// TwinCAT 3 PLC project PISTON_TEST
// ProgramVersion: 3.1.4023.0
// libraries:
//   Tc2_Standard, * (Beckhoff Automation GmbH)
//   Tc2_System, * (Beckhoff Automation GmbH)
//   Tc2_Utilities, * (Beckhoff Automation GmbH)
//   Tc3_Module, * (Beckhoff Automation GmbH)
// project tree:
//   DUTs/ ePistonStatus.TcDUT, E_CONVAYOR_STATE.TcDUT, E_MAIN_STATE.TcDUT, E_PISTON_STATE.TcDUT, E_PISTON_TYPE.TcDUT (not stored), E_STATION_STATE.TcDUT, ST_CART.TcDUT, ST_PISTON.TcDUT
//   GVLs/ GVL.TcGVL
//   / PlcTask.TcTTO
//   POUs/ CLEAN.TcPOU, FB_SEPARATE.TcPOU, MAIN_CONVAYOR.TcPOU, FB_CART.TcPOU, FB_NEW_PISTON.TcPOU, MAIN.TcPOU, PISTONS_CYCLE.TcPOU, SUPPLY.TcPOU, SUPPLY_CONVAYOR.TcPOU (not stored), UpdateTimeStamp.TcPOU (not stored)
// real-time tasks:
//   TASK PlcTask: cycle T#10ms, priority 20, ADS port 350
// motion (NC):
//   TASK NC-Task 1 SAF: cycle T#2ms, priority 4, ADS port 501
//   TASK NC-Task 1 SVB: cycle T#10ms, priority 8, ADS port 511
//   AXIS MAIN (id 1)
//     OtherSettings: AllowMotionCmdToSlave=true
//     encoder EncType=19
//       EncPara: MaxCount=#xffffffff
//     drive DrvType=16
//       DrvPara: MaxCount=#xffffffff, DriveControlDWord=#x00000100
//         Analog: TorqueSetpointScale=10, ScaleFactorActTorque=0.1
//         TimeComp: TaskDelayCycles=1
//     controller CtrType=1
//       CtrPara: PriorControlFactor=1
//         Observer: BandWidth=20
//   AXIS SUPPLY (id 2)
//     OtherSettings: AllowMotionCmdToSlave=true
//     encoder EncType=19
//       EncPara: MaxCount=#xffffffff
//     drive DrvType=16
//       DrvPara: MaxCount=#xffffffff, DriveControlDWord=#x00000100
//         Analog: TorqueSetpointScale=10, ScaleFactorActTorque=0.1
//         TimeComp: TaskDelayCycles=1
//     controller CtrType=1
//       CtrPara: PriorControlFactor=1
//         Observer: BandWidth=20
//   AXIS JACK1 (id 3)
//     OtherSettings: AllowMotionCmdToSlave=true
//     encoder EncType=1
//     drive DrvType=5
//       Analog: TorqueSetpointScale=10, ScaleFactorActTorque=0.1
//       TimeComp: TaskDelayCycles=1
//     controller CtrType=1
//       CtrPara: PriorControlFactor=1
//         Observer: BandWidth=20
//   AXIS JACK2 (id 4)
//     OtherSettings: AllowMotionCmdToSlave=true
//     encoder EncType=1
//     drive DrvType=5
//       Analog: TorqueSetpointScale=10, ScaleFactorActTorque=0.1
//     controller CtrType=1
//       CtrPara: PriorControlFactor=1
//         Observer: BandWidth=20
// I/O:
//   DEVICE Device 3 (EtherCAT), AmsNetId 5.109.70.127.4.1
//     Term 1 (EK1100) [EK1100 EtherCAT Coupler (2A E-Bus)]
//       Term 2 (EL1809) [EL1809 16Ch. Dig. Input 24V, 3ms]
//       Term 10 (EL1809) [EL1809 16Ch. Dig. Input 24V, 3ms]
//       Term 11 (EL1809) [EL1809 16Ch. Dig. Input 24V, 3ms]
//       Term 13 (EL1809) [EL1809 16Ch. Dig. Input 24V, 3ms]
//       Term 3 (EL2869) [EL2869 16Ch. Dig Output 24V, 0.5A, Diagnostic]
//       Term 4 (EL6224) [EL6224 (IO Link Master)]
//       Term 15 (EL9011) [EL9011 End Terminal]
//       Term 7 (EL9011) [EL9011 End Terminal]
//     MAIN
//     SUPPLY [CD02 EtherCAT Drive (CoE)]
// variable links:
//   (this object) <-> Device 3 (EtherCAT)/MAIN
//     Drive/Inputs/In/nDataIn1 <-> TxPDO 1/Following Error Actual Value
//     Drive/Inputs/In/nDataIn3[0] <-> TxPDO 4/Torque Actual Value
//     Drive/Inputs/In/nDcOutputTime <-> InfoData/DcOutputShift
//     Drive/Inputs/In/nState1 <-> TxPDO 4/Statusword
//     Drive/Inputs/In/nState2 <-> TxPDO 4/Statusword @bit 8
//     Drive/Inputs/In/nState4 @bit 1 <-> WcState/InputToggle
//     Drive/Inputs/In/nState4 <-> WcState/WcState
//     Drive/Inputs/In/nState5 <-> TxPDO 3/Modes of Operation Display
//     Drive/Outputs/Out/nCtrl1 <-> RxPDO 4/Controlword
//     Drive/Outputs/Out/nCtrl2 <-> RxPDO 4/Controlword @bit 8
//     Drive/Outputs/Out/nCtrl5 <-> RxPDO 4/Modes of Operation
//     Drive/Outputs/Out/nDataOut1 <-> RxPDO 1/Target Position
//     Drive/Outputs/Out/nDataOut2 <-> RxPDO 2/Target Velocity
//     Drive/Outputs/Out/nDataOut3[0] <-> RxPDO 4/Torque Offset
//     Drive/Outputs/Out/nDataOut4[0] <-> RxPDO 3/Target Torque
//     Enc/Inputs/In/nDataIn1 <-> TxPDO 2/Position Actual Value
//     Enc/Inputs/In/nDcInputTime <-> InfoData/DcInputShift
//     Enc/Inputs/In/nState4 @bit 1 <-> WcState/InputToggle
//     Enc/Inputs/In/nState4 <-> WcState/WcState
//   (this object) <-> Device 3 (EtherCAT)/SUPPLY
//     Drive/Inputs/In/nDataIn1 <-> TxPDO 1/Following Error Actual Value
//     Drive/Inputs/In/nDataIn3[0] <-> TxPDO 4/Torque Actual Value
//     Drive/Inputs/In/nDcOutputTime <-> InfoData/DcOutputShift
//     Drive/Inputs/In/nState1 <-> TxPDO 4/Statusword
//     Drive/Inputs/In/nState2 <-> TxPDO 4/Statusword @bit 8
//     Drive/Inputs/In/nState4 @bit 1 <-> WcState/InputToggle
//     Drive/Inputs/In/nState4 <-> WcState/WcState
//     Drive/Inputs/In/nState5 <-> TxPDO 3/Modes of Operation Display
//     Drive/Outputs/Out/nCtrl1 <-> RxPDO 4/Controlword
//     Drive/Outputs/Out/nCtrl2 <-> RxPDO 4/Controlword @bit 8
//     Drive/Outputs/Out/nCtrl5 <-> RxPDO 4/Modes of Operation
//     Drive/Outputs/Out/nDataOut1 <-> RxPDO 1/Target Position
//     Drive/Outputs/Out/nDataOut2 <-> RxPDO 2/Target Velocity
//     Drive/Outputs/Out/nDataOut3[0] <-> RxPDO 4/Torque Offset
//     Drive/Outputs/Out/nDataOut4[0] <-> RxPDO 3/Target Torque
//     Enc/Inputs/In/nDataIn1 <-> TxPDO 2/Position Actual Value
//     Enc/Inputs/In/nDcInputTime <-> InfoData/DcInputShift
//     Enc/Inputs/In/nState4 @bit 1 <-> WcState/InputToggle
//     Enc/Inputs/In/nState4 <-> WcState/WcState
//   TAMAR_22mm Instance <-> Device 3 (EtherCAT)/Term 1 (EK1100)/Term 2 (EL1809)
//     PlcTask Inputs/GVL_IO.inputs[1]/ch{1..16} <-> Channel {1..16}/ch{1..16}  (16 links)
//   TAMAR_22mm Instance <-> Device 3 (EtherCAT)/Term 1 (EK1100)/Term 3 (EL2869)
//     PlcTask Outputs/GVL_IO.outputs[1]/ch{1..16} <-> DOS Outputs Channel {1..16}/Output  (16 links)
//   TAMAR_22mm Instance <-> Device 3 (EtherCAT)/Term 1 (EK1100)/Term 4 (EL6224)
//     PlcTask Outputs/GVL_IO.uIOLINK1 <-> IO-Link Port1_out/GVL_IO.uIOLINK1
//     PlcTask Outputs/GVL_IO.uIOLINK2 <-> IO-Link Port2_out/GVL_IO.uIOLINK2
//   TAMAR_22mm Instance <-> NC-Task 1 SAF/Axes/JACK1
//     PlcTask Inputs/GVL.Axis_JACK1.Axis.NcToPlc <-> Outputs/ToPlc
//     PlcTask Outputs/GVL.Axis_JACK1.Axis.PlcToNc <-> Inputs/FromPlc
//   TAMAR_22mm Instance <-> NC-Task 1 SAF/Axes/JACK2
//     PlcTask Inputs/GVL.Axis_JACK2.Axis.NcToPlc <-> Outputs/ToPlc
//     PlcTask Outputs/GVL.Axis_JACK2.Axis.PlcToNc <-> Inputs/FromPlc
//   TAMAR_22mm Instance <-> NC-Task 1 SAF/Axes/MAIN
//     PlcTask Inputs/GVL.Axis_MAIN.Axis.NcToPlc <-> Outputs/ToPlc
//     PlcTask Outputs/GVL.Axis_MAIN.Axis.PlcToNc <-> Inputs/FromPlc
//   TAMAR_22mm Instance <-> NC-Task 1 SAF/Axes/SUPPLY
//     PlcTask Inputs/GVL.Axis_SUPPLY.Axis.NcToPlc <-> Outputs/ToPlc
//     PlcTask Outputs/GVL.Axis_SUPPLY.Axis.PlcToNc <-> Inputs/FromPlc

CONFIGURATION PISTON_TEST
    RESOURCE PLC ON TwinCAT3
        TASK PlcTask(INTERVAL := T#10ms, PRIORITY := 20);
        PROGRAM MAIN WITH PlcTask : MAIN;
    END_RESOURCE
END_CONFIGURATION

// ---- DUTs/ePistonStatus.TcDUT
{attribute 'qualified_only'}
{attribute 'strict'}
TYPE ePistonStatus :
(
	OPENED:=0,CLOSED,OPENING,CLOSING,ERROR
);
END_TYPE

// ---- DUTs/E_CONVAYOR_STATE.TcDUT
{attribute 'qualified_only'}
{attribute 'strict'}
TYPE E_CONVAYOR_STATE :
(
	uninit,
	idle,
	do_move,
	done,
	pause,
	error
);
END_TYPE

// ---- DUTs/E_MAIN_STATE.TcDUT
{attribute 'qualified_only'}
{attribute 'strict'}
TYPE E_MAIN_STATE :
(
	uninit,
	idle,
	do_actions,
	move_next,
	done,
	pause,
	error
);
END_TYPE

// ---- DUTs/E_PISTON_STATE.TcDUT
{attribute 'qualified_only'}
{attribute 'strict'}
TYPE E_PISTON_STATE :
(
	init,
	ready,
	busy,
	done,
	error
);
END_TYPE

// ---- DUTs/E_STATION_STATE.TcDUT
{attribute 'qualified_only'}
{attribute 'strict'}
TYPE E_STATION_STATE :
(
	uninit,
	idle,
	do_action1,
	do_action2,
	do_action3,
	do_action4,
	do_action5,
	done,
	pause,
	error
);
END_TYPE

// ---- DUTs/ST_CART.TcDUT
TYPE ST_CART :
STRUCT
	nNAME: STRING;
	posX:INT;
	posY:INT;
	color:INT;
	position: INT;
END_STRUCT
END_TYPE

// ---- DUTs/ST_PISTON.TcDUT
TYPE ST_PISTON :
STRUCT
	ePISTON_TYPE: E_PISTON_TYPE;
	
	nNAME: STRING;
	openTime: REAL:=5;
	closeTime: REAL:=5;
	timeoutOpen:  TIME:=T#5S;
	timeoutClose: TIME:=T#5S;
	bOPEN_BY_DEFAULT: BOOL:= FALSE;
END_STRUCT
	
END_TYPE

// ---- GVLs/GVL.TcGVL
 //{attribute 'qualified_only'}
VAR_GLOBAL
	
	supply_station_num: INT:=1;
	separate1_station_num: INT:=5;
	separate2_station_num: INT:=9;
	clean_station_num: INT:=24;
	total_ready:INT:=0;
	iNUMBER_OF_PISTONS: INT:=15;
	conv_length: INT:=1150;
	conv_height: INT:=290;
	num_of_carts:INT:=18;
	X_OFFSET: INT:=380;
	Y_OFFSET: INT:=352;
	stPISTON_PARAM: ARRAY[1..15] OF  ST_PISTON;
	fbPiston: ARRAY[1..15] OF FB_NEW_PISTON;
	fbCART: ARRAY[1..18] OF FB_CART;
	posArrX:ARRAY[1..36] OF INT;
	posArrY:ARRAY[1..36] OF INT;
	
	eMAIN_STATE: E_MAIN_STATE:= E_MAIN_STATE.uninit;
	eSUPPLY: E_STATION_STATE:=E_STATION_STATE.uninit;
	eSEPARATE1: E_STATION_STATE:=E_STATION_STATE.uninit;
	eSEPARATE2: E_STATION_STATE:=E_STATION_STATE.uninit;
	eCLEAN: E_STATION_STATE:=E_STATION_STATE.uninit;
	eMAIN_CONVAYOR_STATE: E_CONVAYOR_STATE:=E_CONVAYOR_STATE.uninit;
	eSUPPLY_CONVAYOR_STATE: E_CONVAYOR_STATE:=E_CONVAYOR_STATE.uninit;
	
	bSTART: BOOL:=FALSE;// start main state machine
	sup_RUNNING: BOOL:=FALSE;// supply id runing
	clean_RUNNING: BOOL:=FALSE;// cleaning runing
	bS1_RUNNING: BOOL:=FALSE; // station 1 is running
	bS2_RUNNING: BOOL:=FALSE; // station 2 is running
	bCONV_MAIN_INPOS: BOOL:=FALSE; // convayor in position
	bCONV_SUPPLY_INPOS: BOOL:=FALSE; // convayor in position
	bPAUSE_MAIN: BOOL:=FALSE;
	
	
END_VAR

// ---- POUs/MAIN.TcPOU
PROGRAM MAIN
VAR
	counter:INT:=0;
	iNUMBER1 : INT:=2;
	sNAME1 : STRING(255):='24_5A';
	Trigger : BOOL;
	rtrigSTART: R_TRIG;
	rtrigPAUSE: R_TRIG;
	ftrigRERUN: F_TRIG;
	temp_state:E_MAIN_STATE;
	temp_supply_state:E_STATION_STATE;
	temp_sep1_state:E_STATION_STATE;
	temp_sep2_state:E_STATION_STATE;
	temp_clean_state:E_STATION_STATE;
	temp_conv_state:E_CONVAYOR_STATE;
	temp_supconv_state:E_CONVAYOR_STATE;
	
	fbSEPARATION1: FB_SEPARATE;		
	fbSEPARATION2: FB_SEPARATE;	
	
	action_timeout: TON:=(PT:=T#20s);
	move_timeout: TON;
	bTIMEOUT:BOOL:=FALSE;
END_VAR

A_ERROR_CHECK();
PISTONS_CYCLE();
MAIN_CONVAYOR();
SUPPLY_CONVAYOR();
SUPPLY();
fbSEPARATION1(piston_updown:=  fbPiston[3],
			  piston_colet:=  fbPiston[4],
			  piston_puller:=  fbPiston[5],
			  piston_tray:=  fbPiston[6],
			  piston_pins:=  fbPiston[7],
			  eState:= eSEPARATE1 );
		
fbSEPARATION2(piston_updown:=  fbPiston[8],
			  piston_colet:=  fbPiston[9],
			  piston_puller:=  fbPiston[10],
			  piston_tray:=  fbPiston[11],
			  piston_pins:=  fbPiston[12],
			  eState:= eSEPARATE2 );	
	
CLEAN();

rtrigSTART(CLK:= bSTART, Q=> );
rtrigPAUSE(CLK:= bPAUSE_MAIN, Q=> );
ftrigRERUN(CLK:= bPAUSE_MAIN, Q=> );
action_timeout(IN:=bTIMEOUT);

//MAIN_STATE_MACHINE:
CASE eMAIN_STATE OF
	E_MAIN_STATE.uninit:
		bTIMEOUT:=FALSE;
		IF rtrigSTART.Q THEN
			eMAIN_STATE:=E_MAIN_STATE.do_actions;
		END_IF
	
	E_MAIN_STATE.do_actions:
		bTIMEOUT:=TRUE;
		IF eSUPPLY = E_STATION_STATE.idle THEN     
			eSUPPLY := E_STATION_STATE.do_action1;
		END_IF
		IF eSEPARATE1 = E_STATION_STATE.idle THEN
			eSEPARATE1 := E_STATION_STATE.do_action1;
		END_IF
		IF eSEPARATE2 = E_STATION_STATE.idle THEN
			eSEPARATE2 := E_STATION_STATE.do_action1;
		END_IF
		IF eCLEAN = E_STATION_STATE.idle THEN
			eCLEAN := E_STATION_STATE.do_action1;
		END_IF
		
		IF (eSEPARATE1 = E_STATION_STATE.done AND eSEPARATE2 = E_STATION_STATE.done AND eSUPPLY = E_STATION_STATE.done  AND eCLEAN = E_STATION_STATE.done) THEN
			eSUPPLY := E_STATION_STATE.idle;
			eSEPARATE1 := E_STATION_STATE.idle;
			eSEPARATE2 := E_STATION_STATE.idle;
			eCLEAN := E_STATION_STATE.idle;
			eMAIN_STATE:=E_MAIN_STATE.move_next;
			bTIMEOUT:=FALSE;
		END_IF
		
		IF action_timeout.Q THEN
			eMAIN_STATE:=E_MAIN_STATE.error;
		END_IF
		
	E_MAIN_STATE.move_next: 
		IF eMAIN_CONVAYOR_STATE = E_CONVAYOR_STATE.idle THEN
			eMAIN_CONVAYOR_STATE := E_CONVAYOR_STATE.do_move;
		END_IF
		IF eSUPPLY_CONVAYOR_STATE = E_CONVAYOR_STATE.idle THEN
			eSUPPLY_CONVAYOR_STATE := E_CONVAYOR_STATE.do_move;
		END_IF
		IF eMAIN_CONVAYOR_STATE = E_CONVAYOR_STATE.done AND eSUPPLY_CONVAYOR_STATE = E_CONVAYOR_STATE.done THEN
			eMAIN_CONVAYOR_STATE := E_CONVAYOR_STATE.idle;
			eSUPPLY_CONVAYOR_STATE := E_CONVAYOR_STATE.idle;
			eMAIN_STATE:=E_MAIN_STATE.do_actions;
		END_IF
		
	E_MAIN_STATE.pause: 
		bTIMEOUT:=FALSE;
		//paused
		
	E_MAIN_STATE.error: 
		//error mode

END_CASE

IF rtrigPAUSE.Q THEN
	temp_state:=eMAIN_STATE;
	temp_supply_state:=eSUPPLY;
	temp_sep1_state:=eSEPARATE1;
	temp_sep2_state:=eSEPARATE2;
	temp_clean_state:=eCLEAN;
	temp_conv_state:=eMAIN_CONVAYOR_STATE;
	temp_supconv_state:=eMAIN_CONVAYOR_STATE;
	eMAIN_STATE:=E_MAIN_STATE.pause;
	eSUPPLY:=E_STATION_STATE.pause;
	eSEPARATE1:=E_STATION_STATE.pause;
	eSEPARATE2:=E_STATION_STATE.pause;
	eMAIN_CONVAYOR_STATE:=E_CONVAYOR_STATE.pause;
	eSUPPLY_CONVAYOR_STATE:=E_CONVAYOR_STATE.pause;
	
END_IF

IF ftrigRERUN.Q THEN
	eMAIN_STATE:=temp_state;
	eSUPPLY:=temp_supply_state;
	eSEPARATE1:=temp_sep1_state;
	eSEPARATE2:=temp_sep2_state;
	eCLEAN:=temp_clean_state;
	eMAIN_CONVAYOR_STATE:=temp_conv_state;
	eSUPPLY_CONVAYOR_STATE:=temp_conv_state;
END_IF

ACTION A_ERROR_CHECK:
FOR counter:=1 TO iNUMBER_OF_PISTONS BY 1 DO
	IF fbPiston[counter].PistonStatus = ePistonStatus.ERROR THEN
		eMAIN_STATE:=E_MAIN_STATE.error;
		
	END_IF
	
END_FOR;
END_ACTION

END_PROGRAM

// ---- POUs/FB_SEPARATE.TcPOU
FUNCTION_BLOCK FB_SEPARATE
VAR_INPUT
	piston_updown: REFERENCE TO FB_NEW_PISTON;
	piston_colet: REFERENCE TO FB_NEW_PISTON;
	piston_puller: REFERENCE TO FB_NEW_PISTON;
	piston_tray: REFERENCE TO FB_NEW_PISTON;
	piston_pins: REFERENCE TO FB_NEW_PISTON;
	eState: REFERENCE TO  E_STATION_STATE;
END_VAR
VAR_OUTPUT
	bRUNNING:BOOL :=FALSE;
END_VAR
VAR
	tDelay: TON;
	bDELAY: BOOL:=FALSE;
	E: INT;
END_VAR

tDelay(IN:=bDELAY);

CASE eState OF
	E_STATION_STATE.uninit:
		eState:= E_STATION_STATE.idle;

	E_STATION_STATE.idle:
		bRUNNING:=FALSE;
			

	E_STATION_STATE.do_action1://delay and lower device
		bRUNNING:=TRUE;
		tDELAY.PT:=T#0.1S;
		bDELAY:=TRUE;
		IF tDELAY.Q THEN
			bDELAY:=FALSE;
			piston_updown.A_OPEN();
		END_IF
		
		IF piston_updown.PistonStatus= ePistonStatus.OPENED THEN
			eState:=E_STATION_STATE.do_action2;
		END_IF
		
	E_STATION_STATE.do_action2://delay and close colet
		tDELAY.PT:=T#0.1S;
		bDELAY:=TRUE;
		IF tDELAY.Q THEN
			bDELAY:=FALSE;
			piston_colet.A_OPEN();
		END_IF
		
		IF piston_colet.PistonStatus= ePistonStatus.OPENED THEN
			eState:=E_STATION_STATE.do_action3;
		END_IF
	
	E_STATION_STATE.do_action3://delay and pull while raising
		tDELAY.PT:=T#0.2S;		
		bDELAY:=TRUE;
		IF tDELAY.Q THEN
			bDELAY:=FALSE;
			piston_updown.A_CLOSE();
			piston_puller.A_OPEN();
		END_IF
		IF piston_updown.PistonStatus= ePistonStatus.CLOSED AND piston_puller.PistonStatus= ePistonStatus.OPENED THEN
			eState:=E_STATION_STATE.do_action4;
		END_IF
	
	E_STATION_STATE.do_action4://delay close puller and enter tray
		tDELAY.PT:=T#0.2S;		
		bDELAY:=TRUE;
		IF tDELAY.Q THEN
			bDELAY:=FALSE;
			piston_puller.A_CLOSE();
			piston_tray.A_OPEN();
		END_IF
		IF piston_puller.PistonStatus= ePistonStatus.CLOSED AND piston_tray.PistonStatus= ePistonStatus.OPENED THEN
			eState:=E_STATION_STATE.do_action5;
		END_IF

	E_STATION_STATE.do_action5://release colet and push pins
		tDELAY.PT:=T#0.2S;		
		bDELAY:=TRUE;
		IF tDELAY.Q THEN
			bDELAY:=FALSE;
			piston_colet.A_CLOSE();
			piston_pins.A_OPEN();
		END_IF
		IF piston_colet.PistonStatus= ePistonStatus.CLOSED AND piston_pins.PistonStatus= ePistonStatus.OPENED THEN
			eState:=E_STATION_STATE.do_action6;
		END_IF
		
	E_STATION_STATE.do_action6://raise pins and close tray
		tDELAY.PT:=T#0.2S;		
		bDELAY:=TRUE;
		IF tDELAY.Q THEN
			bDELAY:=FALSE;
			piston_pins.A_CLOSE();
			piston_tray.A_CLOSE();
		END_IF
		IF piston_colet.PistonStatus= ePistonStatus.CLOSED AND piston_pins.PistonStatus= ePistonStatus.CLOSED THEN
			eState:=E_STATION_STATE.do_action7;
		END_IF	
		
	E_STATION_STATE.do_action7://delay
		tDELAY.PT:=T#0.1S;
		bDELAY:=TRUE;
		IF tDELAY.Q THEN
			bDELAY:=FALSE;
			eState:=E_STATION_STATE.done;
		END_IF
		
	
	E_STATION_STATE.done:
		bRUNNING:=FALSE;
		
	E_STATION_STATE.pause:
		//paused

END_CASE

END_FUNCTION_BLOCK

// ---- POUs/FB_NEW_PISTON.TcPOU
FUNCTION_BLOCK FB_NEW_PISTON
VAR_INPUT
	
	bMANUAL:BOOL:=FALSE;
	stPISTON:   ST_PISTON;
	bCMD_OPEN_SWR: BOOL;
	bCMD_CLOSE_SWR: BOOL;
	bCMD_OPEN: BOOL;
	bSEN_OPEN: BOOL;
	bSEN_CLOSE: BOOL;
END_VAR
VAR_OUTPUT
	PistonStatus:ePistonStatus;
	bVALVE_OPEN: BOOL;
	bVALVE_CLOSE: BOOL;
	
	
END_VAR
VAR
	timerOpening:ton;
	timerClosing:ton;
	timeoutOpening:ton;
	timeoutClosing:ton;
	bSTARTUP: BOOL:=FALSE;
	
	
END_VAR

   IF NOT bSTARTUP THEN
	bCMD_OPEN:=stPISTON.bOPEN_BY_DEFAULT;
	bSTARTUP:=TRUE;
END_IF

timerOpening(IN:= bVALVE_OPEN, PT:=REAL_TO_TIME(stPISTON.openTime)*1000 , Q=> , ET=> );
timerClosing(IN:= NOT bVALVE_OPEN, PT:=REAL_TO_TIME(stPISTON.closeTime)*1000 , Q=> , ET=> );
timeoutOpening(IN:= bVALVE_OPEN AND NOT bSEN_OPEN, PT:= stPISTON.timeoutOpen, Q=> , ET=> );
timeoutClosing(IN:= NOT bVALVE_OPEN AND NOT bSEN_CLOSE, PT:= stPISTON.timeoutClose, Q=> , ET=> );
IF bMANUAL THEN
	bVALVE_OPEN:= bCMD_OPEN;
	bVALVE_CLOSE:= NOT bCMD_OPEN;
ELSE
	bVALVE_OPEN:= bCMD_OPEN_SWR;
	bVALVE_CLOSE:= NOT bCMD_OPEN_SWR;
END_IF



CASE stPISTON.ePISTON_TYPE OF
	0://NO_SENSORS
		IF bVALVE_OPEN AND NOT timerOpening.Q THEN
			PistonStatus:=ePistonStatus.OPENING;
		ELSIF bVALVE_OPEN AND timerOpening.Q THEN
			PistonStatus:=ePistonStatus.OPENED;
		ELSIF bVALVE_CLOSE AND NOT timerClosing.Q THEN
			PistonStatus:=ePistonStatus.CLOSING;
		ELSIF bVALVE_CLOSE AND timerClosing.Q THEN
			PistonStatus:=ePistonStatus.CLOSED;
		END_IF
		
 
	
	1://only open sensor
	
		IF bVALVE_OPEN AND NOT bSEN_OPEN THEN
			PistonStatus:=ePistonStatus.OPENING;
		ELSIF bVALVE_OPEN AND bSEN_OPEN THEN
			PistonStatus:=ePistonStatus.OPENED;
		ELSIF bVALVE_CLOSE AND NOT timerClosing.Q THEN
			PistonStatus:=ePistonStatus.CLOSING;
		ELSIF bVALVE_CLOSE AND timerClosing.Q THEN
			PistonStatus:=ePistonStatus.CLOSED;
		END_IF
	
	2:// only close sensor
		IF bVALVE_OPEN AND NOT timerOpening.Q THEN
			PistonStatus:=ePistonStatus.OPENING;
		ELSIF bVALVE_OPEN AND timerOpening.Q THEN
			PistonStatus:=ePistonStatus.OPENED;
		ELSIF bVALVE_CLOSE AND NOT bSEN_CLOSE THEN
			PistonStatus:=ePistonStatus.CLOSING;
		ELSIF bVALVE_CLOSE AND bSEN_CLOSE THEN
			PistonStatus:=ePistonStatus.CLOSED;
		END_IF
	
	
	3://both sensors
		IF bVALVE_OPEN AND NOT bSEN_OPEN THEN
			PistonStatus:=ePistonStatus.OPENING;
		ELSIF bVALVE_OPEN AND bSEN_OPEN THEN
			PistonStatus:=ePistonStatus.OPENED;
		ELSIF bVALVE_CLOSE AND NOT bSEN_CLOSE THEN
			PistonStatus:=ePistonStatus.CLOSING;
		ELSIF bVALVE_CLOSE AND bSEN_CLOSE THEN
			PistonStatus:=ePistonStatus.CLOSED;
		END_IF
	
END_CASE

IF timeoutOpening.Q AND (stPISTON.ePISTON_TYPE = E_PISTON_TYPE.ONLY_OPEN OR stPISTON.ePISTON_TYPE = E_PISTON_TYPE.BOTH)  THEN
	PistonStatus:=ePistonStatus.ERROR;
END_IF
IF timeoutClosing.Q  AND (stPISTON.ePISTON_TYPE = E_PISTON_TYPE.ONLY_CLOSE OR stPISTON.ePISTON_TYPE = E_PISTON_TYPE.BOTH)  THEN
	PistonStatus:=ePistonStatus.ERROR;
END_IF

ACTION A_CLOSE:
bCMD_OPEN_SWR:=FALSE;
END_ACTION

ACTION A_OPEN:
bCMD_OPEN_SWR:=TRUE;
END_ACTION

END_FUNCTION_BLOCK

// ---- POUs/PISTONS_CYCLE.TcPOU
PROGRAM PISTONS_CYCLE
VAR
	
	bSTARTUP: BOOL:=FALSE;
	counter: INT;
	
END_VAR

IF NOT bSTARTUP THEN
	
	stPISTON_PARAM[1].nNAME:='SUPPLY 1';
	stPISTON_PARAM[1].bOPEN_BY_DEFAULT:=FALSE;
	stPISTON_PARAM[1].openTime:=0.2;
	stPISTON_PARAM[1].closeTime:=0.2;
	stPISTON_PARAM[1].timeoutOpen:=T#3S;
	stPISTON_PARAM[1].timeoutClose:=T#3S;
	stPISTON_PARAM[1].ePISTON_TYPE:= 0;

	stPISTON_PARAM[2].nNAME:='SUPPLY2';
	stPISTON_PARAM[2].bOPEN_BY_DEFAULT:=FALSE;
	stPISTON_PARAM[2].openTime:=0.2;
	stPISTON_PARAM[2].closeTime:=0.2;
	stPISTON_PARAM[2].timeoutOpen:=T#2S;
	stPISTON_PARAM[2].timeoutClose:=T#2S;
	stPISTON_PARAM[2].ePISTON_TYPE:= 0;

	stPISTON_PARAM[3].nNAME:='SEPARATE1 UP_DOWN';
	stPISTON_PARAM[3].bOPEN_BY_DEFAULT:=FALSE;
	stPISTON_PARAM[3].openTime:=0.2;
	stPISTON_PARAM[3].closeTime:=0.2;
	stPISTON_PARAM[3].timeoutOpen:=T#3S;
	stPISTON_PARAM[3].timeoutClose:=T#3S;
	stPISTON_PARAM[3].ePISTON_TYPE:= 0;
	
	stPISTON_PARAM[4].nNAME:='SEPARATE1 COLET';
	stPISTON_PARAM[4].bOPEN_BY_DEFAULT:=FALSE;
	stPISTON_PARAM[4].openTime:=0.2;
	stPISTON_PARAM[4].closeTime:=0.2;
	stPISTON_PARAM[4].timeoutOpen:=T#3S;
	stPISTON_PARAM[4].timeoutClose:=T#3S;
	stPISTON_PARAM[4].ePISTON_TYPE:= 0;
	
	stPISTON_PARAM[5].nNAME:='SEPARATE1 PULL';
	stPISTON_PARAM[5].bOPEN_BY_DEFAULT:=FALSE;
	stPISTON_PARAM[5].openTime:=0.2;
	stPISTON_PARAM[5].closeTime:=0.2;
	stPISTON_PARAM[5].timeoutOpen:=T#3S;
	stPISTON_PARAM[5].timeoutClose:=T#3S;
	stPISTON_PARAM[5].ePISTON_TYPE:= 0;
	
	stPISTON_PARAM[6].nNAME:='SEPARATE1 TRAY';
	stPISTON_PARAM[6].bOPEN_BY_DEFAULT:=FALSE;
	stPISTON_PARAM[6].openTime:=0.2;
	stPISTON_PARAM[6].closeTime:=0.2;
	stPISTON_PARAM[6].timeoutOpen:=T#3S;
	stPISTON_PARAM[6].timeoutClose:=T#3S;
	stPISTON_PARAM[6].ePISTON_TYPE:= 0;
	
	stPISTON_PARAM[7].nNAME:='SEPARATE1 PINS';
	stPISTON_PARAM[7].bOPEN_BY_DEFAULT:=FALSE;
	stPISTON_PARAM[7].openTime:=0.2;
	stPISTON_PARAM[7].closeTime:=0.2;
	stPISTON_PARAM[7].timeoutOpen:=T#3S;
	stPISTON_PARAM[7].timeoutClose:=T#3S;
	stPISTON_PARAM[7].ePISTON_TYPE:= 0;
	
	stPISTON_PARAM[8].nNAME:='SEPARATE2 UP_DOWN';
	stPISTON_PARAM[8].bOPEN_BY_DEFAULT:=FALSE;
	stPISTON_PARAM[8].openTime:=0.2;
	stPISTON_PARAM[8].closeTime:=0.2;
	stPISTON_PARAM[8].timeoutOpen:=T#3S;
	stPISTON_PARAM[8].timeoutClose:=T#3S;
	stPISTON_PARAM[8].ePISTON_TYPE:= 0;
	
	stPISTON_PARAM[9].nNAME:='SEPARATE2 GRIP';
	stPISTON_PARAM[9].bOPEN_BY_DEFAULT:=FALSE;
	stPISTON_PARAM[9].openTime:=0.2;
	stPISTON_PARAM[9].closeTime:=0.2;
	stPISTON_PARAM[9].timeoutOpen:=T#3S;
	stPISTON_PARAM[9].timeoutClose:=T#3S;
	stPISTON_PARAM[9].ePISTON_TYPE:= 0;
	
	stPISTON_PARAM[10].nNAME:='SEPARATE2 PULL';
	stPISTON_PARAM[10].bOPEN_BY_DEFAULT:=FALSE;
	stPISTON_PARAM[10].openTime:=0.2;
	stPISTON_PARAM[10].closeTime:=0.2;
	stPISTON_PARAM[10].timeoutOpen:=T#3S;
	stPISTON_PARAM[10].timeoutClose:=T#3S;
	stPISTON_PARAM[10].ePISTON_TYPE:= 0;
	
	stPISTON_PARAM[11].nNAME:='SEPARATE2 TRAY';
	stPISTON_PARAM[11].bOPEN_BY_DEFAULT:=FALSE;
	stPISTON_PARAM[11].openTime:=0.2;
	stPISTON_PARAM[11].closeTime:=0.2;
	stPISTON_PARAM[11].timeoutOpen:=T#3S;
	stPISTON_PARAM[11].timeoutClose:=T#3S;
	stPISTON_PARAM[11].ePISTON_TYPE:= 0;
	
	stPISTON_PARAM[12].nNAME:='SEPARATE2 PINS';
	stPISTON_PARAM[12].bOPEN_BY_DEFAULT:=FALSE;
	stPISTON_PARAM[12].openTime:=0.2;
	stPISTON_PARAM[12].closeTime:=0.2;
	stPISTON_PARAM[12].timeoutOpen:=T#3S;
	stPISTON_PARAM[12].timeoutClose:=T#3S;
	stPISTON_PARAM[12].ePISTON_TYPE:= 0;
	
	stPISTON_PARAM[13].nNAME:='ADVANCE';
	stPISTON_PARAM[13].bOPEN_BY_DEFAULT:=FALSE;
	stPISTON_PARAM[13].openTime:=0.5;
	stPISTON_PARAM[13].closeTime:=0.5;
	stPISTON_PARAM[13].timeoutOpen:=T#3S;
	stPISTON_PARAM[13].timeoutClose:=T#3S;
	stPISTON_PARAM[13].ePISTON_TYPE:= 0;
	
	stPISTON_PARAM[14].nNAME:='CLEAN';
	stPISTON_PARAM[14].bOPEN_BY_DEFAULT:=FALSE;
	stPISTON_PARAM[14].openTime:=0.2;
	stPISTON_PARAM[14].closeTime:=0.2;
	stPISTON_PARAM[14].timeoutOpen:=T#3S;
	stPISTON_PARAM[14].timeoutClose:=T#3S;
	stPISTON_PARAM[14].ePISTON_TYPE:= 0;
	
	FOR counter:=1 TO iNUMBER_OF_PISTONS BY 1 DO
		fbPiston[counter](stPISTON:=stPISTON_PARAM[counter]);
	END_FOR;
	
	bSTARTUP:=TRUE;
END_IF
FOR counter:=1 TO iNUMBER_OF_PISTONS BY 1 DO
	fbPiston[counter]();
END_FOR;

END_PROGRAM

// ---- POUs/SUPPLY.TcPOU
PROGRAM SUPPLY
VAR

	tDelay: TON;
	bDELAY: BOOL:=FALSE;
END_VAR

tDelay(IN:=bDELAY);
CASE eSUPPLY OF
	E_STATION_STATE.uninit:
		eSUPPLY:= E_STATION_STATE.idle;

	E_STATION_STATE.idle:
		bS1_RUNNING:=FALSE;
			

	E_STATION_STATE.do_action1://delay and open piston1,2
		tDELAY.PT:=T#1S;
		bDELAY:=TRUE;
		IF tDELAY.Q THEN
			bDELAY:=FALSE;
			fbPISTON[1].A_OPEN();
			fbPISTON[2].A_OPEN();
		END_IF
		
		IF fbPISTON[1].PistonStatus= ePistonStatus.OPENED  AND fbPISTON[2].PistonStatus= ePistonStatus.OPENED THEN
			eSUPPLY:=E_STATION_STATE.do_action2;
		END_IF
		
	E_STATION_STATE.do_action2://delay and close pistons 1,2
		tDELAY.PT:=T#2S;		
		bDELAY:=TRUE;
		IF tDELAY.Q THEN
			bDELAY:=FALSE;
			fbPISTON[1].A_CLOSE();
			fbPISTON[2].A_CLOSE();
		END_IF
		IF fbPISTON[1].PistonStatus= ePistonStatus.CLOSED  AND fbPISTON[2].PistonStatus= ePistonStatus.CLOSED THEN
			eSUPPLY:=E_STATION_STATE.do_action5;
		END_IF
	
	E_STATION_STATE.do_action3://delay and open piston 3
		//...
	
	E_STATION_STATE.do_action4://delay and close pistons 1,2
		//...
		
	E_STATION_STATE.do_action5://delay 
		tDELAY.PT:=T#2S;
		bDELAY:=TRUE;
		IF tDELAY.Q THEN
			bDELAY:=FALSE;
			eSUPPLY:=E_STATION_STATE.done;
		END_IF
	
	E_STATION_STATE.done:
		bS1_RUNNING:=FALSE;
		
	E_STATION_STATE.pause:
		//paused

END_CASE

END_PROGRAM

// ---- POUs/CLEAN.TcPOU
PROGRAM CLEAN
VAR
	tDelay: TON;
	bDELAY: BOOL:=FALSE;
END_VAR

tDelay(IN:=bDELAY);
CASE eCLEAN OF
	E_STATION_STATE.uninit:
		eCLEAN:= E_STATION_STATE.idle;

	E_STATION_STATE.idle:
		clean_RUNNING:=FALSE;
			

	E_STATION_STATE.do_action1://delay and open piston8
		clean_RUNNING:=TRUE;
		tDELAY.PT:=T#0.3S;
		bDELAY:=TRUE;
		IF tDELAY.Q THEN
			bDELAY:=FALSE;
			fbPISTON[14].A_OPEN();
		END_IF
		
		IF fbPISTON[14].PistonStatus= ePistonStatus.OPENED THEN
			eCLEAN:=E_STATION_STATE.do_action2;
		END_IF
		
	
	
	E_STATION_STATE.do_action2://delay and close pistons 8
		tDELAY.PT:=T#1S;		
		bDELAY:=TRUE;
		IF tDELAY.Q THEN
			bDELAY:=FALSE;
			fbPISTON[14].A_CLOSE();
		END_IF
		IF fbPISTON[14].PistonStatus= ePistonStatus.CLOSED  THEN
			eCLEAN:=E_STATION_STATE.do_action3;
		END_IF
	
	E_STATION_STATE.do_action3://delay
		tDELAY.PT:=T#1S;
		bDELAY:=TRUE;
		IF tDELAY.Q THEN
			bDELAY:=FALSE;
			eCLEAN:=E_STATION_STATE.done;
		END_IF
		
	
	E_STATION_STATE.done:
		clean_RUNNING:=FALSE;
		
	E_STATION_STATE.pause:
		//paused

END_CASE

END_PROGRAM

// ---- POUs/MAIN_CONVAYOR.TcPOU
PROGRAM MAIN_CONVAYOR
VAR
	inc: INT:=1;
	temp: INT;
	state: INT:=0;
	total_length: INT;
	cart_space: INT;
	cornerX: INT;
	cornerY: INT;
	bMOVE:BOOL :=FALSE;
	bSTARTUP: BOOL:=FALSE;
	rtrigNext: R_TRIG;
	counter: INT;
	tNext: TON;
	tDelay: TON;
	bDELAY: BOOL:=FALSE;
	first_run: BOOL:=FALSE;
END_VAR

FOR counter:=1 TO num_of_carts BY 1 DO
	fbCART[counter]();
END_FOR;

IF NOT first_run THEN
	A_set_cart_spaces();
	A_SETUP();
	first_run:=TRUE;
END_IF



tDelay(IN:=bDELAY);
tNext(IN:=bMOVE , PT:=T#1S , Q=> , ET=> );

CASE eMAIN_CONVAYOR_STATE OF
	E_CONVAYOR_STATE.uninit:
		A_SETUP();
		eMAIN_CONVAYOR_STATE:=E_CONVAYOR_STATE.idle;
	
	E_CONVAYOR_STATE.idle:
		bDELAY:=FALSE;
		bMOVE:=FALSE;
		bCONV_MAIN_INPOS:=TRUE;
	
	E_CONVAYOR_STATE.do_move: // open advance piston and update carts
		IF bCONV_MAIN_INPOS THEN		 
			A_CARTS_STEP();
			fbPISTON[11].A_OPEN();
			bCONV_MAIN_INPOS:=FALSE;
		END_IF
		bMOVE:=TRUE;
		bCONV_MAIN_INPOS:=FALSE;
		IF fbPISTON[11].PistonStatus= ePistonStatus.OPENED THEN
			A_CARTS_STEP();
			bMOVE:=FALSE;
			bCONV_MAIN_INPOS:=TRUE;
			eMAIN_CONVAYOR_STATE:=E_CONVAYOR_STATE.st1;
		END_IF
	
	E_CONVAYOR_STATE.st1://delay and close advansed piston
		tDELAY.PT:=T#0.6S;
		bDELAY:=TRUE;
		IF tDelay.Q THEN
			fbPISTON[11].A_CLOSE();
			eMAIN_CONVAYOR_STATE:=E_CONVAYOR_STATE.done;
		END_IF
		IF fbPISTON[11].PistonStatus= ePistonStatus.CLOSED THEN
			//...
		END_IF		
	
	E_CONVAYOR_STATE.done:
		//...
	
	E_CONVAYOR_STATE.pause:
	//paused
	
END_CASE

ACTION A_CARTS_STEP:
FOR counter:=1 TO num_of_carts BY 1 DO
	fbCART[counter].A_STEP();
END_FOR;
END_ACTION

ACTION A_set_cart_spaces:
 total_length := (conv_height*2)+(conv_length*2);
cart_space := total_length /((num_of_carts*2));
inc:=1;
posArrX[inc]:= 0+X_OFFSET;
posArrY[inc]:= 0+(conv_height/2)+Y_OFFSET;



WHILE state = 0 DO    //left1
	IF posArrY[inc]-cart_space < Y_OFFSET THEN
		temp :=cart_space - (posArrY[inc]-Y_OFFSET);
		posArrX[inc+1]:= temp+X_OFFSET;
		posArrY[inc+1]:= 0+Y_OFFSET;
		state:=1;
	ELSE
		posArrX[inc+1]:= 0+X_OFFSET;
		posArrY[inc+1]:=posArrY[inc]- cart_space;
		inc :=inc+1;
	END_IF
END_WHILE
inc := inc+1;

WHILE state = 1 DO // top
	IF posArrX[inc]+cart_space > (X_OFFSET+conv_length) THEN
		temp :=cart_space - ((X_OFFSET+conv_length)-posArrX[inc]);
		posArrX[inc+1]:= conv_length+X_OFFSET;
		posArrY[inc+1]:= temp+Y_OFFSET;
		state:=2;
	ELSE
		posArrX[inc+1]:= posArrX[inc]+cart_space;
		posArrY[inc+1]:=Y_OFFSET;
		inc :=inc+1;
	END_IF
END_WHILE
inc :=inc+1;	

WHILE state = 2 DO // right
	IF posArrY[inc]+cart_space > (Y_OFFSET+conv_height) THEN
		temp :=cart_space - ((Y_OFFSET+conv_height)-posArrY[inc]);
		posArrX[inc+1]:= (conv_length+X_OFFSET)-temp;
		posArrY[inc+1]:= 0+Y_OFFSET+conv_height;
		state:=3;
	ELSE
		posArrX[inc+1]:= 0+X_OFFSET+conv_length;
		posArrY[inc+1]:=posArrY[inc]+ cart_space;
		inc :=inc+1;
	END_IF	
END_WHILE
inc :=inc+1;	

WHILE state = 3 DO //bottom
	IF  posArrX[inc]-cart_space < X_OFFSET THEN
		temp :=cart_space - (posArrX[inc]-X_OFFSET);
		posArrX[inc+1]:= X_OFFSET;
		posArrY[inc+1]:= Y_OFFSET+ conv_height-temp;
		state:=4;
	ELSE
		posArrX[inc+1]:= posArrX[inc]-cart_space;
		posArrY[inc+1]:=Y_OFFSET+conv_height;
		inc :=inc+1;
		
	END_IF
END_WHILE

IF inc > 34 THEN
	RETURN;
END_IF


inc :=inc+1;

WHILE state = 4 DO    //left2
	IF posArrY[inc]-cart_space < ((conv_height/2)+Y_OFFSET) THEN
		state:=5;
	ELSE
		posArrX[inc+1]:= 0+X_OFFSET;
		posArrY[inc+1]:=posArrY[inc]- cart_space;
		inc :=inc+1;
		
	END_IF
END_WHILE
END_ACTION

ACTION A_SETUP:
	bSTARTUP:=TRUE;
	fbCART[1].stCART.position:=1;
	fbCART[1].stCART.color:=1;
	fbCART[1].stCART.nNAME:=INT_TO_STRING(1001);
	fbCART[1].stCART.posX:=posArrX[1];
	fbCART[1].stCART.posY:=posArrY[1];
		
	FOR counter:=1 TO (num_of_carts-1) BY 1 DO
		fbCART[counter+1].stCART.position:=37-((counter*2));
		fbCART[counter+1].stCART.color:=1;
		fbCART[counter+1].stCART.nNAME:=INT_TO_STRING(1000+counter+1);
		fbCART[counter+1].stCART.posX:=posArrX[37-((counter*2))];
		fbCART[counter+1].stCART.posY:=posArrY[37-((counter*2))];
	END_FOR;
END_ACTION

END_PROGRAM

// ---- POUs/FB_CART.TcPOU
FUNCTION_BLOCK FB_CART
VAR_INPUT
	stCART: ST_CART;
END_VAR
VAR_OUTPUT
END_VAR

VAR
	inner_counter: INT;
END_VAR

ACTION A_STEP:
IF stCART.position < num_of_carts*2 THEN
	stCART.position:= stCART.position+1;
	stCART.posX:=posArrX[stCART.position];
	stCART.posY:=posArrY[stCART.position];
ELSE
	stCART.position:= 1;
	stCART.posX:=posArrX[stCART.position];
	stCART.posY:=posArrY[stCART.position];
	
END_IF
END_ACTION

END_FUNCTION_BLOCK
